TYPE ST_ClosedLoopParams :
STRUCT
	fProportionalGain: LREAL;
	fIntegralGain: LREAL;
	fMaxAllowableError : LREAL; 
END_STRUCT
END_TYPE

(* stored: Version 1.1.0.1, ProductVersion 3.1.4024.12
   DUT ST_ClosedLoopParams: Id {02b16262-2b47-4e8d-87cd-7a161db0bb2f} *)
